Fanuc KAREL source: NC0087.KL

-- PROVISIONAL review KL for V1013-1; original PC SHA256 4fe0bb10ccc625040b761f29a19523a90fab5046491e2cce0f1cc572204b5323
-- Incomplete behavior may be omitted. Consult companion uncertainty JSON. Do not deploy.
PROGRAM NC0087
%NOLOCKGROUP
-- UNRESOLVED_LOCAL_POOL 3 cells at code offset 3; source declarations unknown
-- DIRECT_LOCAL_WORD_ACCESS alone does not prove INTEGER, REAL, or BOOLEAN
BEGIN
  -- UNRESOLVED_PC offsets 0-8; opcodes 2B,2C,7B
  -- UNRESOLVED_PC offsets 13-20; opcodes 9D,23
  -- UNRESOLVED_PC offsets 25-38; opcodes 21,9D,57,79
  -- UNRESOLVED_PC offsets 43-60; opcodes 21,40,41,42
  -- UNRESOLVED_PC offsets 65-94; opcodes 9D,23,9E,2E,22,7A
  -- UNRESOLVED_PC offsets 99-116; opcodes 21,2E,59,79
  -- UNRESOLVED_PC offsets 121-134; opcodes 21,9D,57,79
  -- UNRESOLVED_PC offsets 139-156; opcodes 21,40,41,42
  -- UNRESOLVED_PC offsets 161-190; opcodes 9D,23,9E,2E,22,7A
  -- UNRESOLVED_PC offsets 195-212; opcodes 21,2E,59,79
  -- UNRESOLVED_PC offsets 217-230; opcodes 21,9D,57,79
  -- UNRESOLVED_PC offsets 235-252; opcodes 21,40,41,42
  -- UNRESOLVED_PC offsets 257-287; opcodes 21,9D,52,23,7A,40,41,42
  -- UNRESOLVED_PC offsets 292-316; opcodes 21,2E,52,23,7A,43
  -- UNRESOLVED_PC offsets 321-339; opcodes 21,2E,52,23
  -- UNRESOLVED_PC offsets 349-354; opcodes 7A
  -- UNRESOLVED_PC offsets 359-377; opcodes 21,2E,52,23
  -- UNRESOLVED_PC offsets 387-392; opcodes 7A
  -- UNRESOLVED_PC offsets 397-428; opcodes 20,2C,23,7A,40,41,42
  -- UNRESOLVED_PC offsets 433-457; opcodes 21,2E,52,23,7A,43
  -- UNRESOLVED_PC offsets 462-480; opcodes 21,2E,52,23
  -- UNRESOLVED_PC offsets 490-495; opcodes 7A
  -- UNRESOLVED_PC offsets 500-518; opcodes 21,2E,52,23
  -- UNRESOLVED_PC offsets 528-533; opcodes 7A
  -- UNRESOLVED_PC offsets 538-569; opcodes 20,2C,23,7A,40,41,42
  -- UNRESOLVED_PC offsets 574-598; opcodes 21,2E,52,23,7A,43
  -- UNRESOLVED_PC offsets 603-621; opcodes 21,2E,52,23
  -- UNRESOLVED_PC offsets 631-636; opcodes 7A
  -- UNRESOLVED_PC offsets 641-659; opcodes 21,2E,52,23
  -- UNRESOLVED_PC offsets 669-673; opcodes 7F
  -- UNRESOLVED_PC offsets 678-682; opcodes 27,AA
  -- UNRESOLVED_PC offsets 687-691; opcodes 7F
END NC0087
